TYPE ST_CommandHistoryEntry :
STRUCT
    dtTrigger: DT;
    dtRelease: DT;
    dtFinish: DT;
    fVelocity: LREAL;
    fAcceleration: LREAL;
    fDeceleration: LREAL;
    fPosition: LREAL;
    eCommand: E_MotionFunctions := E_MotionFunctions.eWaitingForCommand;
    eResult: E_Result := E_Result.eNone;
END_STRUCT
END_TYPE

(* stored: Version 1.1.0.1
   DUT ST_CommandHistoryEntry: Id {b7472ac7-f553-0458-2fb0-2b71a79014f5} *)
